Yaskawa INFORM job: OK_R2_O51(P)(180,0_50)AWOK.JBI

/JOB
//NAME OK_R2_O51(P)(180,0_50)AWOK
///FOLDERNAME X4
//POS
///NPOS 171,171,171,7,0,0
///TOOL 0
///POSTYPE PULSE
///PULSE
C00000=-50858,-152082,-121144,18649,17915,51634
C00001=-147168,-149464,-118878,19599,23894,51283
C00002=-161827,-134621,-107268,25398,3105,50110
C00003=-145259,-126792,-102407,-35778,11198,78058
C00004=-116021,-129119,-97228,-53911,31006,88799
C00005=-125899,-119752,-73479,23033,53920,53167
C00006=-125735,-114890,-67549,23322,52814,52975
C00007=-125671,-112960,-65155,23449,52353,52891
C00008=-126105,-110187,-62624,23598,52349,52699
C00009=-125671,-112960,-65155,23449,52353,52891
C00010=-118903,-119552,-66906,23649,51064,55199
C00011=-116388,-115921,-66848,21286,56152,54864
C00012=-114859,-123419,-67349,21635,45840,56131
C00013=-114872,-125580,-69766,21507,46195,56212
C00014=-114905,-131076,-75767,21222,47015,56394
C00015=-128675,-128885,-89754,22399,59592,53270
C00016=-128484,-124084,-84033,22588,58564,53127
C00017=-128409,-122195,-81734,22673,58133,53064
C00018=-128859,-120120,-79518,22852,57980,52843
C00019=-128409,-122195,-81734,22673,58133,53064
C00020=-114682,-125524,-89732,18708,67552,56611
C00021=-115293,-123846,-88718,19749,69071,59080
C00022=-110984,-145278,-91981,19087,48630,58517
C00023=-110973,-147767,-94346,19033,48794,58556
C00024=-110946,-154290,-100276,18941,49070,58624
C00025=-126969,-138385,-101497,26913,69331,54689
C00026=-125925,-134718,-96194,27021,67761,54719
C00027=-125507,-133245,-94058,27071,67127,54730
C00028=-126132,-131351,-92377,27159,67271,54516
C00029=-125507,-133245,-94058,27071,67127,54730
C00030=-115086,-147474,-96729,26876,58765,56850
C00031=-113078,-148944,-96555,26779,57371,57323
C00032=-115086,-147474,-96729,26876,58765,56850
C00033=-115592,-149500,-98985,26865,59233,56762
C00034=-116854,-154731,-104630,26862,60331,56524
C00035=-125864,-146646,-114501,37777,34164,45574
C00036=-123511,-186562,-123386,24932,18534,8837
C00037=-117479,-144936,-115289,-27220,31518,-36752
C00038=-114583,-111112,-67320,-30996,68419,-79803
C00039=-118450,-109814,-63048,-31301,65358,-80470
C00040=-120054,-109187,-61290,-31423,64137,-80759
C00041=-120065,-106918,-59050,-31475,63950,-80705
C00042=-120054,-109187,-61290,-31423,64137,-80759
C00043=-121189,-120165,-62504,-32737,59555,-79778
C00044=-121208,-121946,-61698,-33188,58355,-79378
C00045=-121189,-120165,-62504,-32737,59555,-79778
C00046=-119205,-121057,-64365,-32572,60842,-79373
C00047=-114458,-123027,-68910,-32135,64047,-78441
C00048=-115872,-117575,-82827,-29920,73365,-81695
C00049=-119572,-116939,-78927,-30035,70257,-82326
C00050=-121103,-116552,-77315,-30079,69029,-82602
C00051=-121101,-114825,-75467,-30125,68813,-82541
C00052=-121103,-116552,-77315,-30079,69029,-82602
C00053=-119821,-145601,-89258,-31809,62933,-80293
C00054=-119755,-148274,-88828,-32255,61557,-79832
C00055=-119821,-145601,-89258,-31809,62933,-80293
C00056=-117714,-146483,-91028,-31707,64224,-79826
C00057=-112701,-148366,-95356,-31403,67459,-78765
C00058=-115324,-128295,-94676,-31217,76358,-79594
C00059=-119104,-128105,-90959,-31349,73084,-80184
C00060=-120676,-127869,-89415,-31402,71795,-80449
C00061=-120677,-126314,-88026,-31410,71747,-80436
C00062=-120676,-127869,-89415,-31402,71795,-80449
C00063=-120434,-145492,-92931,-32753,65996,-78610
C00064=-120414,-147161,-92365,-33041,64984,-78279
C00065=-120434,-145492,-92931,-32753,65996,-78610
C00066=-118477,-146193,-94638,-32637,67304,-78214
C00067=-113816,-147586,-98796,-32315,70592,-77322
C00068=-120568,-139125,-94129,-37659,61084,-32062
C00069=-120567,-135030,-88943,-38024,60216,-31717
C00070=-120562,-135623,-87366,-38473,59204,-31306
C00071=-120564,-135572,-88662,-38181,59857,-31572
C00072=-120553,-135497,-86870,-38563,59018,-31224
C00073=-120564,-135211,-87266,-38419,59325,-31356
C00074=-120567,-135085,-88951,-38032,60197,-31710
C00075=-120568,-139184,-94137,-37667,61063,-32054
C00076=-120568,-139242,-94145,-37676,61043,-32046
C00077=-120567,-135139,-88958,-38041,60178,-31702
C00078=-122131,-135263,-87277,-38235,58637,-31815
C00079=-120564,-135680,-88675,-38198,59820,-31557
C00080=-120553,-135602,-86882,-38580,58981,-31209
C00081=-120563,-135010,-87213,-38394,59377,-31378
C00082=-120567,-135194,-88965,-38049,60159,-31695
C00083=-120568,-139301,-94153,-37684,61023,-32038
C00084=-120565,-129876,-82142,-38569,58996,-31221
C00085=-120564,-125889,-76861,-39020,58049,-30823
C00086=-121805,-125856,-75053,-39322,56656,-30820
C00087=-120561,-126316,-76545,-39180,57725,-30684
C00088=-120551,-126068,-74668,-39590,56926,-30333
C00089=-139324,-123913,-74595,-35947,49925,-36615
C00090=-120564,-125936,-76867,-39027,58033,-30817
C00091=-120565,-129925,-82148,-38577,58979,-31213
C00092=-120565,-129776,-82130,-38553,59031,-31235
C00093=-120564,-125796,-76851,-39004,58082,-30837
C00094=-122348,-126275,-75206,-39308,56329,-30941
C00095=-120561,-126223,-76535,-39164,57758,-30698
C00096=-120551,-125978,-74659,-39574,56957,-30347
C00097=-139614,-124103,-74665,-35903,49767,-36691
C00098=-120564,-125843,-76856,-39012,58065,-30830
C00099=-120565,-129826,-82136,-38561,59013,-31228
C00100=-120438,-148134,-72436,-40343,44873,-27172
C00101=-120436,-142644,-66735,-40792,44345,-26886
C00102=-120422,-141711,-64519,-41392,43675,-26507
C00103=-120427,-142724,-66211,-41036,44070,-26730
C00104=-120399,-141589,-63928,-41601,43455,-26370
C00105=-120420,-141724,-64512,-41397,43666,-26503
C00106=-120436,-142676,-66731,-40805,44330,-26878
C00107=-120438,-148169,-72431,-40356,44857,-27163
C00108=-120562,-116904,-64691,-40188,55809,-29841
C00109=-120561,-112917,-59184,-40780,54776,-29365
C00110=-120557,-112485,-57242,-41229,54034,-29012
C00111=-120547,-112748,-56806,-41422,53730,-28860
C00112=-120563,-109425,-55080,-41116,54215,-29101
C00113=-120558,-112218,-57172,-41186,54104,-29047
C00114=-120561,-112955,-59188,-40788,54763,-29359
C00115=-120562,-116944,-64695,-40196,55795,-29834
C00116=-117479,-144936,-115289,-27220,31518,-36752
C00117=-123511,-186562,-123386,24932,18534,8837
C00118=-125864,-146646,-114501,37777,34164,45574
C00119=-120568,-139571,-94039,19597,41682,51990
C00120=-120567,-135434,-88842,20008,40670,51744
C00121=-120566,-134209,-86850,20248,40107,51603
C00122=-118862,-135262,-86623,19504,39068,52248
C00123=-119974,-135747,-88507,19806,40185,51935
C00124=-121182,-134915,-87023,20715,40018,51252
C00125=-120567,-135402,-88849,20000,40689,51749
C00126=-120568,-139536,-94045,19589,41702,51995
C00127=-120568,-139501,-94051,19581,41723,52000
C00128=-120567,-135370,-88856,19992,40709,51754
C00129=-120180,-134104,-86854,19998,40069,51798
C00130=-118864,-135201,-86637,19488,39107,52257
C00131=-119975,-135684,-88521,19790,40224,51944
C00132=-120947,-135143,-87103,20605,39895,51345
C00133=-120567,-135338,-88862,19984,40728,51758
C00134=-120568,-139466,-94057,19573,41743,52005
C00135=-120565,-130131,-82013,20615,39280,51388
C00136=-120564,-126118,-76724,21141,38162,51085
C00137=-120237,-125281,-74483,21383,37193,50991
C00138=-118859,-125745,-74402,20657,36590,51593
C00139=-119972,-126347,-76360,20936,37697,51282
C00140=-120628,-125475,-74602,21636,37268,50796
C00141=-120564,-126091,-76732,21132,38179,51090
C00142=-120565,-130102,-82020,20607,39298,51393
C00143=-120565,-130188,-81998,20631,39244,51379
C00144=-120564,-126171,-76707,21158,38127,51076
C00145=-120353,-125325,-74544,21448,37235,50939
C00146=-118857,-125795,-74384,20673,36555,51584
C00147=-119971,-126399,-76344,20952,37663,51273
C00148=-120721,-125521,-74505,21734,37212,50728
C00149=-120564,-126144,-76716,21149,38144,51080
C00150=-120565,-130159,-82005,20623,39262,51383
C00151=-120562,-119389,-67536,14587,38107,53162
C00152=-120561,-115341,-62001,15025,36823,52914
C00153=-120561,-113908,-59765,15249,36205,52790
C00154=-118851,-114725,-59512,14375,35359,53549
C00155=-119967,-115470,-61579,14771,36406,53150
C00156=-120560,-114223,-59902,15275,36129,52774
C00157=-120561,-115320,-62011,15019,36840,52918
C00158=-120562,-119366,-67545,14581,38124,53165
C00159=-120562,-119343,-67555,14575,38141,53169
C00160=-120561,-115299,-62021,15013,36856,52921
C00161=-120560,-114241,-59922,15276,36132,52776
C00162=-118853,-114685,-59532,14364,35391,53554
C00163=-119968,-115429,-61599,14760,36439,53156
C00164=-120677,-114417,-59979,15368,36101,52704
C00165=-120561,-115277,-62031,15008,36872,52924
C00166=-120562,-119320,-67564,14570,38158,53172
C00167=-120518,-162682,-102707,14754,37514,53074
C00168=-120518,-162682,-102707,14754,37514,53074
C00169=-120518,-162817,-102707,14754,-6597,53074
C00170=7651,-162817,-102707,14754,-6597,53074
BC00000=188697,682303,1064074
BC00001=186165,685733,1061366
BC00002=167778,742292,1047372
BC00003=167817,755862,1049853
BC00004=167902,785869,1055340
BC00005=168210,894343,1075175
BC00006=168210,894343,1075175
BC00007=168210,894343,1075175
BC00008=168210,894343,1075175
BC00009=168210,894343,1075175
BC00010=168210,894343,1075175
BC00011=168210,894343,1075175
BC00012=168210,894343,1075175
BC00013=168210,894343,1075175
BC00014=168210,894343,1075175
BC00015=197697,861884,1075175
BC00016=197697,861884,1075175
BC00017=197697,861884,1075175
BC00018=197697,861884,1075175
BC00019=197697,861884,1075175
BC00020=197697,861884,1075175
BC00021=197697,861884,1075175
BC00022=197697,861884,1075175
BC00023=197697,861884,1075175
BC00024=197697,861884,1075175
BC00025=204756,850926,1075175
BC00026=204756,850926,1075175
BC00027=204756,850926,1075175
BC00028=204756,850926,1075175
BC00029=204756,850926,1075175
BC00030=204756,850926,1075175
BC00031=204756,850926,1075175
BC00032=204756,850926,1075175
BC00033=204756,850926,1075175
BC00034=204756,850926,1075175
BC00035=168210,813037,1075175
BC00036=228943,832659,1075175
BC00037=329672,865204,1075175
BC00038=337121,951989,1075175
BC00039=337121,951989,1075175
BC00040=337121,951989,1075175
BC00041=337121,951989,1075175
BC00042=337121,951989,1075175
BC00043=337121,951989,1075175
BC00044=337121,951989,1075175
BC00045=337121,951989,1075175
BC00046=337121,951989,1075175
BC00047=337121,951989,1075175
BC00048=337862,907687,1075175
BC00049=337862,907687,1075175
BC00050=337862,907687,1075175
BC00051=337862,907687,1075175
BC00052=337862,907687,1075175
BC00053=337862,907687,1075175
BC00054=337862,907687,1075175
BC00055=337862,907687,1075175
BC00056=337862,907687,1075175
BC00057=337862,907687,1075175
BC00058=340309,878845,1075175
BC00059=340309,878845,1075175
BC00060=340309,878845,1075175
BC00061=340309,878845,1075175
BC00062=340309,878845,1075175
BC00063=340309,878845,1075175
BC00064=340309,878845,1075175
BC00065=340309,878845,1075175
BC00066=340309,878845,1075175
BC00067=340309,878845,1075175
BC00068=361841,856908,1075175
BC00069=360454,859447,1075175
BC00070=359900,860463,1075175
BC00071=359900,860463,1075175
BC00072=359900,860463,1075175
BC00073=343972,860415,1075175
BC00074=344527,859399,1075175
BC00075=345913,856860,1075175
BC00076=329985,856812,1075175
BC00077=328599,859351,1075175
BC00078=328044,860367,1075175
BC00079=328044,860367,1075175
BC00080=328044,860367,1075175
BC00081=312116,860319,1075175
BC00082=312671,859303,1075175
BC00083=314058,856764,1075175
BC00084=329884,891305,1075175
BC00085=328498,893845,1075175
BC00086=327943,894860,1075175
BC00087=327943,894860,1075175
BC00088=327943,894860,1075175
BC00089=327943,894860,1075175
BC00090=312570,893797,1075175
BC00091=313957,891257,1075175
BC00092=361740,891401,1075175
BC00093=360353,893940,1075175
BC00094=359799,894956,1075175
BC00095=359799,894956,1075175
BC00096=359799,894956,1075175
BC00097=359799,894956,1075175
BC00098=344426,893893,1075175
BC00099=345812,891353,1075175
BC00100=351733,962185,1075175
BC00101=351036,964755,1075175
BC00102=350757,965784,1075175
BC00103=350757,965784,1075175
BC00104=350757,965784,1075175
BC00105=334829,965736,1075175
BC00106=335108,964707,1075175
BC00107=335806,962137,1075175
BC00108=329672,931452,1075175
BC00109=328286,933991,1075175
BC00110=327731,935007,1075175
BC00111=327731,935007,1075175
BC00112=327731,935007,1075175
BC00113=311961,934959,1075175
BC00114=312516,933943,1075175
BC00115=313902,931404,1075175
BC00116=329672,865204,1075175
BC00117=228943,832659,1075175
BC00118=168210,813037,1075175
BC00119=203914,800542,1075175
BC00120=203285,803344,1075175
BC00121=203034,804465,1075175
BC00122=203034,804465,1075175
BC00123=203034,804465,1075175
BC00124=215203,814376,1075175
BC00125=215455,813255,1075175
BC00126=216084,810452,1075175
BC00127=228253,820363,1075175
BC00128=227624,823165,1075175
BC00129=227373,824286,1075175
BC00130=227373,824286,1075175
BC00131=227373,824286,1075175
BC00132=239538,834194,1075175
BC00133=239794,833076,1075175
BC00134=240423,830273,1075175
BC00135=205215,846714,1075175
BC00136=204586,849516,1075175
BC00137=204334,850637,1075175
BC00138=204334,850637,1075175
BC00139=204334,850637,1075175
BC00140=216504,860548,1075175
BC00141=216755,859427,1075175
BC00142=217384,856625,1075175
BC00143=180876,826893,1075175
BC00144=180247,829695,1075175
BC00145=179995,830816,1075175
BC00146=179995,830816,1075175
BC00147=179995,830816,1075175
BC00148=192165,840727,1075175
BC00149=192416,839606,1075175
BC00150=193045,836804,1075175
BC00151=162569,862636,1075175
BC00152=161394,865032,1075175
BC00153=160924,865991,1075175
BC00154=160924,865991,1075175
BC00155=160924,865991,1075175
BC00156=173094,875901,1075175
BC00157=173564,874943,1075175
BC00158=174738,872546,1075175
BC00159=186908,882457,1075175
BC00160=185733,884853,1075175
BC00161=185263,885812,1075175
BC00162=185263,885812,1075175
BC00163=185263,885812,1075175
BC00164=197428,895718,1075175
BC00165=197903,894764,1075175
BC00166=199077,892367,1075175
BC00167=199077,892367,1075175
BC00168=199077,834176,1075175
BC00169=199077,834176,1075175
BC00170=199077,668242,1075175
EC00000=1596313,309217
EC00001=1596313,309233
EC00002=1596312,309313
EC00003=1596312,309299
EC00004=1596312,309267
EC00005=1596313,309153
EC00006=1596313,309153
EC00007=1596313,309153
EC00008=1596313,309153
EC00009=1596313,309153
EC00010=1596313,309153
EC00011=1596313,309153
EC00012=1596313,309153
EC00013=1596313,309153
EC00014=1596313,309153
EC00015=1596313,309153
EC00016=1596313,309153
EC00017=1596313,309153
EC00018=1596313,309153
EC00019=1596313,309153
EC00020=1596313,309153
EC00021=1596313,309153
EC00022=1596313,309153
EC00023=1596313,309153
EC00024=1596313,309153
EC00025=1596313,309153
EC00026=1596313,309153
EC00027=1596313,309153
EC00028=1596313,309153
EC00029=1596313,309153
EC00030=1596313,309153
EC00031=1596313,309153
EC00032=1596313,309153
EC00033=1596313,309153
EC00034=1596313,309153
EC00035=1596313,309153
EC00036=1596313,402182
EC00037=1596313,556475
EC00038=1596313,556475
EC00039=1596313,556475
EC00040=1596313,556475
EC00041=1596313,556475
EC00042=1596313,556475
EC00043=1596313,556475
EC00044=1596313,556475
EC00045=1596313,556475
EC00046=1596313,556475
EC00047=1596313,556475
EC00048=1596313,556475
EC00049=1596313,556475
EC00050=1596313,556475
EC00051=1596313,556475
EC00052=1596313,556475
EC00053=1596313,556475
EC00054=1596313,556475
EC00055=1596313,556475
EC00056=1596313,556475
EC00057=1596313,556475
EC00058=1596313,556475
EC00059=1596313,556475
EC00060=1596313,556475
EC00061=1596313,556475
EC00062=1596313,556475
EC00063=1596313,556475
EC00064=1596313,556475
EC00065=1596313,556475
EC00066=1596313,556475
EC00067=1596313,556475
EC00068=1596313,556475
EC00069=1596313,556475
EC00070=1596313,556475
EC00071=1596313,556475
EC00072=1596313,556475
EC00073=1596313,556475
EC00074=1596313,556475
EC00075=1596313,556475
EC00076=1596313,556475
EC00077=1596313,556475
EC00078=1596313,556475
EC00079=1596313,556475
EC00080=1596313,556475
EC00081=1596313,556475
EC00082=1596313,556475
EC00083=1596313,556475
EC00084=1596313,556475
EC00085=1596313,556475
EC00086=1596313,556475
EC00087=1596313,556475
EC00088=1596313,556475
EC00089=1596313,556475
EC00090=1596313,556475
EC00091=1596313,556475
EC00092=1596313,556475
EC00093=1596313,556475
EC00094=1596313,556475
EC00095=1596313,556475
EC00096=1596313,556475
EC00097=1596313,556475
EC00098=1596313,556475
EC00099=1596313,556475
EC00100=1596313,556475
EC00101=1596313,556475
EC00102=1596313,556475
EC00103=1596313,556475
EC00104=1596313,556475
EC00105=1596313,556475
EC00106=1596313,556475
EC00107=1596313,556475
EC00108=1596313,556475
EC00109=1596313,556475
EC00110=1596313,556475
EC00111=1596313,556475
EC00112=1596313,556475
EC00113=1596313,556475
EC00114=1596313,556475
EC00115=1596313,556475
EC00116=1596313,556475
EC00117=1596313,402182
EC00118=1596313,309153
EC00119=1596313,309153
EC00120=1596313,309153
EC00121=1596313,309153
EC00122=1596313,309153
EC00123=1596313,309153
EC00124=1596313,309153
EC00125=1596313,309153
EC00126=1596313,309153
EC00127=1596313,309153
EC00128=1596313,309153
EC00129=1596313,309153
EC00130=1596313,309153
EC00131=1596313,309153
EC00132=1596313,309153
EC00133=1596313,309153
EC00134=1596313,309153
EC00135=1596313,309153
EC00136=1596313,309153
EC00137=1596313,309153
EC00138=1596313,309153
EC00139=1596313,309153
EC00140=1596313,309153
EC00141=1596313,309153
EC00142=1596313,309153
EC00143=1596313,309153
EC00144=1596313,309153
EC00145=1596313,309153
EC00146=1596313,309153
EC00147=1596313,309153
EC00148=1596313,309153
EC00149=1596313,309153
EC00150=1596313,309153
EC00151=1596313,309153
EC00152=1596313,309153
EC00153=1596313,309153
EC00154=1596313,309153
EC00155=1596313,309153
EC00156=1596313,309153
EC00157=1596313,309153
EC00158=1596313,309153
EC00159=1596313,309153
EC00160=1596313,309153
EC00161=1596313,309153
EC00162=1596313,309153
EC00163=1596313,309153
EC00164=1596313,309153
EC00165=1596313,309153
EC00166=1596313,309153
EC00167=1596313,309153
EC00168=1596313,309153
EC00169=1596313,309153
EC00170=1596313,309153
///POSTYPE BASE
///RECTAN
///RCONF 0,0,0,0,0,0,0,0,0,0,0,0,0,0,0,0,0,0,0,0,0,0,0,0
P00006=0.222,-3.123,-1.508,0.0000,0.0000,0.0000
P00021=-0.225,-6.128,-0.405,0.0000,0.0000,0.0000
P00022=0.222,-3.123,-1.508,0.0000,0.0000,0.0000
P00023=0.143,-0.036,0.682,0.0000,0.0000,0.0000
P00031=1.853,-0.001,-1.549,0.0000,0.0000,0.0000
P00032=1.957,0.503,-7.217,0.0000,0.0000,0.0000
///RCONF 0,0,0,0,1,0,0,0,0,0,0,0,0,0,0,0,0,0,0,0,0,0,0,0
P00033=-0.123,0.612,-5.012,0.0000,0.0000,0.0000
//INST
///DATE 2023/12/14 18:46
///ATTR SC,RW
///GROUP1 RB1,BS1
///GROUP2 ST1
NOP
'OK_r2_O51(P)(180,0_50)
'180,50
'Path S1557
SFTOF3D
MOVJ C00000 BC00000 VJ=50.00  +MOVJ EC00000 VJ=50.00
MOVJ C00001 BC00001 VJ=50.00  +MOVJ EC00001 VJ=50.00
MOVJ C00002 BC00002 VJ=50.00  +MOVJ EC00002 VJ=50.00
MOVJ C00003 BC00003 VJ=50.00  +MOVJ EC00003 VJ=50.00
MOVJ C00004 BC00004 VJ=50.00  +MOVJ EC00004 VJ=50.00
MOVJ C00005 BC00005 VJ=100.00  +MOVJ EC00005 VJ=100.00
MOVL C00006 BC00006 V=100.0  +MOVJ EC00006 VJ=100.00
SMOVL C00007 BC00007 V=60.0  +MOVJ EC00007
SREFP 3 C00008 BC00008  +REFP EC00008
CALL JOB:SEARCH-R1-S13D
SET P021 P006
SFTON3D P021
SMOVL C00009 BC00009 V=60.0  +MOVJ EC00009
SMOVL C00010 BC00010 V=60.0  +MOVJ EC00010
SREFP 3 C00011 BC00011  +REFP EC00011
CALL JOB:SEARCH-R1-S13D
SET P021 P006
SFTON3D P021
SMOVL C00012 BC00012 V=60.0  +MOVJ EC00012
MOVL C00013 BC00013 V=400.0  +MOVJ EC00013 VJ=100.00
MOVL C00014 BC00014 V=1000.0  +MOVJ EC00014 VJ=100.00
'Path S1558
SFTOF3D
MOVJ C00015 BC00015 VJ=100.00  +MOVJ EC00015 VJ=100.00
MOVL C00016 BC00016 V=100.0  +MOVJ EC00016 VJ=100.00
SMOVL C00017 BC00017 V=60.0  +MOVJ EC00017
SREFP 3 C00018 BC00018  +REFP EC00018
CALL JOB:SEARCH-R1-S13D
SET P022 P006
SFTON3D P022
SMOVL C00019 BC00019 V=60.0  +MOVJ EC00019
SMOVL C00020 BC00020 V=60.0  +MOVJ EC00020
SREFP 3 C00021 BC00021  +REFP EC00021
CALL JOB:SEARCH-R1-S13D
SET P022 P006
SFTON3D P022
SMOVL C00022 BC00022 V=60.0  +MOVJ EC00022
MOVL C00023 BC00023 V=400.0  +MOVJ EC00023 VJ=100.00
MOVL C00024 BC00024 V=1000.0  +MOVJ EC00024 VJ=100.00
'Path S1559
SFTOF3D
MOVJ C00025 BC00025 VJ=100.00  +MOVJ EC00025 VJ=100.00
MOVL C00026 BC00026 V=100.0  +MOVJ EC00026 VJ=100.00
SMOVL C00027 BC00027 V=60.0  +MOVJ EC00027
SREFP 3 C00028 BC00028  +REFP EC00028
CALL JOB:SEARCH-R1-S13D
SET P023 P006
SFTON3D P023
SMOVL C00029 BC00029 V=60.0  +MOVJ EC00029
SMOVL C00030 BC00030 V=60.0  +MOVJ EC00030
SREFP 3 C00031 BC00031  +REFP EC00031
CALL JOB:SEARCH-R1-S13D
SET P023 P006
SFTON3D P023
SMOVL C00032 BC00032 V=60.0  +MOVJ EC00032
MOVL C00033 BC00033 V=400.0  +MOVJ EC00033 VJ=100.00
MOVL C00034 BC00034 V=1000.0  +MOVJ EC00034 VJ=100.00
MOVJ C00035 BC00035 VJ=100.00  +MOVJ EC00035 VJ=100.00
MOVJ C00036 BC00036 VJ=100.00  +MOVJ EC00036 VJ=100.00
MOVJ C00037 BC00037 VJ=100.00  +MOVJ EC00037 VJ=100.00
'180,0
'Path S1123
SFTOF3D
MOVJ C00038 BC00038 VJ=100.00  +MOVJ EC00038 VJ=100.00
MOVL C00039 BC00039 V=400.0  +MOVJ EC00039 VJ=100.00
SMOVL C00040 BC00040 V=60.0  +MOVJ EC00040
SREFP 3 C00041 BC00041  +REFP EC00041
CALL JOB:SEARCH-R1-S13D
SET P031 P006
SFTON3D P031
SMOVL C00042 BC00042 V=60.0  +MOVJ EC00042
SMOVL C00043 BC00043 V=60.0  +MOVJ EC00043
SREFP 3 C00044 BC00044  +REFP EC00044
CALL JOB:SEARCH-R1-S13D
SET P031 P006
SFTON3D P031
SMOVL C00045 BC00045 V=60.0  +MOVJ EC00045
MOVL C00046 BC00046 V=400.0  +MOVJ EC00046 VJ=100.00
MOVL C00047 BC00047 V=1000.0  +MOVJ EC00047 VJ=100.00
'Path S1130
SFTOF3D
MOVJ C00048 BC00048 VJ=100.00  +MOVJ EC00048 VJ=100.00
MOVL C00049 BC00049 V=400.0  +MOVJ EC00049 VJ=100.00
SMOVL C00050 BC00050 V=60.0  +MOVJ EC00050
SREFP 3 C00051 BC00051  +REFP EC00051
CALL JOB:SEARCH-R1-S13D
SET P032 P006
SFTON3D P032
SMOVL C00052 BC00052 V=60.0  +MOVJ EC00052
SMOVL C00053 BC00053 V=60.0  +MOVJ EC00053
SREFP 3 C00054 BC00054  +REFP EC00054
CALL JOB:SEARCH-R1-S13D
SET P032 P006
SFTON3D P032
SMOVL C00055 BC00055 V=60.0  +MOVJ EC00055
MOVL C00056 BC00056 V=400.0  +MOVJ EC00056 VJ=100.00
MOVL C00057 BC00057 V=1000.0  +MOVJ EC00057 VJ=100.00
'Path S1131
SFTOF3D
MOVJ C00058 BC00058 VJ=100.00  +MOVJ EC00058 VJ=100.00
MOVL C00059 BC00059 V=400.0  +MOVJ EC00059 VJ=100.00
SMOVL C00060 BC00060 V=60.0  +MOVJ EC00060
SREFP 3 C00061 BC00061  +REFP EC00061
CALL JOB:SEARCH-R1-S13D
SET P033 P006
SFTON3D P033
SMOVL C00062 BC00062 V=60.0  +MOVJ EC00062
SMOVL C00063 BC00063 V=60.0  +MOVJ EC00063
SREFP 3 C00064 BC00064  +REFP EC00064
CALL JOB:SEARCH-R1-S13D
SET P033 P006
SFTON3D P033
SMOVL C00065 BC00065 V=60.0  +MOVJ EC00065
MOVL C00066 BC00066 V=400.0  +MOVJ EC00066 VJ=100.00
MOVL C00067 BC00067 V=1000.0  +MOVJ EC00067 VJ=100.00
SFTOF3D
'Path W348
SFTOF3D
SFTON3D P033
MOVJ C00068 BC00068 VJ=100.00  +MOVJ EC00068 VJ=100.00
SMOVL C00069 BC00069 V=400.0  +MOVJ EC00069
SMOVL C00070 BC00070 V=100.0 PL=0  +MOVJ EC00070
SREFP 1 C00071 BC00071  +REFP EC00071
SREFP 2 C00072 BC00072  +REFP EC00072
MACRO1 MJ#(0) ARGF0
ARCON
SMOVL C00073 BC00073 V=10.0  +MOVJ EC00073
ARCOF
SMOVL C00074 BC00074 V=400.0  +MOVJ EC00074
SMOVL C00075 BC00075 V=1000.0  +MOVJ EC00075
SFTOF3D
'Path W349
SFTOF3D
SFTON3D P033
MOVJ C00076 BC00076 VJ=100.00  +MOVJ EC00076 VJ=100.00
SMOVL C00077 BC00077 V=400.0  +MOVJ EC00077
SMOVL C00078 BC00078 V=100.0 PL=0  +MOVJ EC00078
SREFP 1 C00079 BC00079  +REFP EC00079
SREFP 2 C00080 BC00080  +REFP EC00080
MACRO1 MJ#(0) ARGF0
ARCON
SMOVL C00081 BC00081 V=10.0  +MOVJ EC00081
ARCOF
SMOVL C00082 BC00082 V=400.0  +MOVJ EC00082
SMOVL C00083 BC00083 V=1000.0  +MOVJ EC00083
SFTOF3D
'Path W350
SFTOF3D
SFTON3D P032
MOVJ C00084 BC00084 VJ=100.00  +MOVJ EC00084 VJ=100.00
SMOVL C00085 BC00085 V=400.0  +MOVJ EC00085
SMOVL C00086 BC00086 V=100.0 PL=0  +MOVJ EC00086
SREFP 1 C00087 BC00087  +REFP EC00087
SREFP 2 C00088 BC00088  +REFP EC00088
MACRO1 MJ#(0) ARGF0
ARCON
SMOVL C00089 BC00089 V=10.0  +MOVJ EC00089
ARCOF
SMOVL C00090 BC00090 V=400.0  +MOVJ EC00090
SMOVL C00091 BC00091 V=1000.0  +MOVJ EC00091
SFTOF3D
'Path W351
SFTOF3D
SFTON3D P032
MOVJ C00092 BC00092 VJ=100.00  +MOVJ EC00092 VJ=100.00
SMOVL C00093 BC00093 V=400.0  +MOVJ EC00093
SMOVL C00094 BC00094 V=100.0 PL=0  +MOVJ EC00094
SREFP 1 C00095 BC00095  +REFP EC00095
SREFP 2 C00096 BC00096  +REFP EC00096
MACRO1 MJ#(0) ARGF0
ARCON
SMOVL C00097 BC00097 V=10.0  +MOVJ EC00097
ARCOF
SMOVL C00098 BC00098 V=400.0  +MOVJ EC00098
SMOVL C00099 BC00099 V=1000.0  +MOVJ EC00099
SFTOF3D
'Path W1132
SFTOF3D
SFTON3D P031
MOVJ C00100 BC00100 VJ=100.00  +MOVJ EC00100 VJ=100.00
SMOVL C00101 BC00101 V=400.0  +MOVJ EC00101
SMOVL C00102 BC00102 V=100.0 PL=0  +MOVJ EC00102
SREFP 1 C00103 BC00103  +REFP EC00103
SREFP 2 C00104 BC00104  +REFP EC00104
MACRO1 MJ#(0) ARGF0
ARCON
SMOVL C00105 BC00105 V=10.0  +MOVJ EC00105
ARCOF
SMOVL C00106 BC00106 V=400.0  +MOVJ EC00106
SMOVL C00107 BC00107 V=1000.0  +MOVJ EC00107
SFTOF3D
'Path W1133
SFTOF3D
SFTON3D P031
MOVJ C00108 BC00108 VJ=100.00  +MOVJ EC00108 VJ=100.00
SMOVL C00109 BC00109 V=400.0  +MOVJ EC00109
SMOVL C00110 BC00110 V=100.0 PL=0  +MOVJ EC00110
SREFP 1 C00111 BC00111  +REFP EC00111
SREFP 2 C00112 BC00112  +REFP EC00112
MACRO1 MJ#(0) ARGF0
ARCON
SMOVL C00113 BC00113 V=10.0  +MOVJ EC00113
ARCOF
SMOVL C00114 BC00114 V=400.0  +MOVJ EC00114
SMOVL C00115 BC00115 V=1000.0  +MOVJ EC00115
SFTOF3D
MOVJ C00116 BC00116 VJ=100.00  +MOVJ EC00116 VJ=100.00
MOVJ C00117 BC00117 VJ=100.00  +MOVJ EC00117 VJ=100.00
MOVJ C00118 BC00118 VJ=100.00  +MOVJ EC00118 VJ=100.00
'180,50
SFTOF3D
'Path W1560
SFTOF3D
SFTON3D P023
MOVJ C00119 BC00119 VJ=100.00  +MOVJ EC00119 VJ=100.00
SMOVL C00120 BC00120 V=100.0  +MOVJ EC00120
SMOVL C00121 BC00121 V=100.0 PL=0  +MOVJ EC00121
SREFP 1 C00122 BC00122  +REFP EC00122
SREFP 2 C00123 BC00123  +REFP EC00123
MACRO1 MJ#(0) ARGF0
ARCON
SMOVL C00124 BC00124 V=10.0  +MOVJ EC00124
ARCOF
SMOVL C00125 BC00125 V=400.0  +MOVJ EC00125
SMOVL C00126 BC00126 V=1000.0  +MOVJ EC00126
SFTOF3D
'Path W1561
SFTOF3D
SFTON3D P023
MOVJ C00127 BC00127 VJ=100.00  +MOVJ EC00127 VJ=100.00
SMOVL C00128 BC00128 V=100.0  +MOVJ EC00128
SMOVL C00129 BC00129 V=100.0 PL=0  +MOVJ EC00129
SREFP 1 C00130 BC00130  +REFP EC00130
SREFP 2 C00131 BC00131  +REFP EC00131
MACRO1 MJ#(0) ARGF0
ARCON
SMOVL C00132 BC00132 V=10.0  +MOVJ EC00132
ARCOF
SMOVL C00133 BC00133 V=400.0  +MOVJ EC00133
SMOVL C00134 BC00134 V=1000.0  +MOVJ EC00134
SFTOF3D
'Path W1562
SFTOF3D
SFTON3D P022
MOVJ C00135 BC00135 VJ=100.00  +MOVJ EC00135 VJ=100.00
SMOVL C00136 BC00136 V=100.0  +MOVJ EC00136
SMOVL C00137 BC00137 V=100.0 PL=0  +MOVJ EC00137
SREFP 1 C00138 BC00138  +REFP EC00138
SREFP 2 C00139 BC00139  +REFP EC00139
MACRO1 MJ#(0) ARGF0
ARCON
SMOVL C00140 BC00140 V=10.0  +MOVJ EC00140
ARCOF
SMOVL C00141 BC00141 V=400.0  +MOVJ EC00141
SMOVL C00142 BC00142 V=1000.0  +MOVJ EC00142
SFTOF3D
'Path W1563
SFTOF3D
SFTON3D P022
MOVJ C00143 BC00143 VJ=100.00  +MOVJ EC00143 VJ=100.00
SMOVL C00144 BC00144 V=100.0  +MOVJ EC00144
SMOVL C00145 BC00145 V=100.0 PL=0  +MOVJ EC00145
SREFP 1 C00146 BC00146  +REFP EC00146
SREFP 2 C00147 BC00147  +REFP EC00147
MACRO1 MJ#(0) ARGF0
ARCON
SMOVL C00148 BC00148 V=10.0  +MOVJ EC00148
ARCOF
SMOVL C00149 BC00149 V=400.0  +MOVJ EC00149
SMOVL C00150 BC00150 V=1000.0  +MOVJ EC00150
SFTOF3D
'Path W1564
SFTOF3D
SFTON3D P021
MOVJ C00151 BC00151 VJ=100.00  +MOVJ EC00151 VJ=100.00
SMOVL C00152 BC00152 V=100.0  +MOVJ EC00152
SMOVL C00153 BC00153 V=100.0 PL=0  +MOVJ EC00153
SREFP 1 C00154 BC00154  +REFP EC00154
SREFP 2 C00155 BC00155  +REFP EC00155
MACRO1 MJ#(0) ARGF0
ARCON
SMOVL C00156 BC00156 V=10.0  +MOVJ EC00156
ARCOF
SMOVL C00157 BC00157 V=400.0  +MOVJ EC00157
SMOVL C00158 BC00158 V=1000.0  +MOVJ EC00158
SFTOF3D
'Path W1565
SFTOF3D
SFTON3D P021
MOVJ C00159 BC00159 VJ=100.00  +MOVJ EC00159 VJ=100.00
SMOVL C00160 BC00160 V=100.0  +MOVJ EC00160
SMOVL C00161 BC00161 V=100.0 PL=0  +MOVJ EC00161
SREFP 1 C00162 BC00162  +REFP EC00162
SREFP 2 C00163 BC00163  +REFP EC00163
MACRO1 MJ#(0) ARGF0
ARCON
SMOVL C00164 BC00164 V=10.0  +MOVJ EC00164
ARCOF
SMOVL C00165 BC00165 V=400.0  +MOVJ EC00165
SMOVL C00166 BC00166 V=1000.0  +MOVJ EC00166
SFTOF3D
MOVJ C00167 BC00167 VJ=50.00  +MOVJ EC00167 VJ=50.00
MOVJ C00168 BC00168 VJ=50.00  +MOVJ EC00168 VJ=50.00
MOVJ C00169 BC00169 VJ=50.00  +MOVJ EC00169 VJ=50.00
MOVJ C00170 BC00170 VJ=50.00  +MOVJ EC00170 VJ=50.00
END
